Universal Robots PolyScope program: Programa_PickPlace.urp

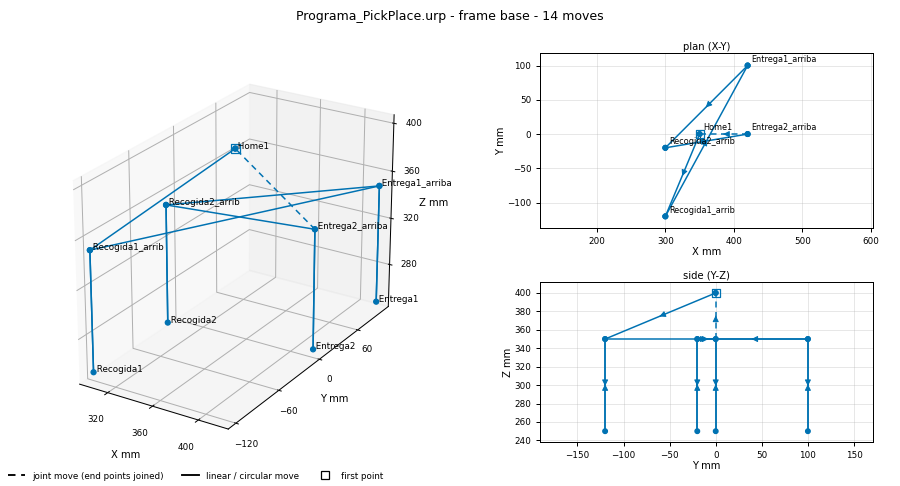
[picture p0: tool path of Programa_PickPlace.urp in frame base, 14 of 14 moves have a stored position in this frame; points joined in program order, loops and branches not executed]
Program Programa_PickPlace (installation=lab_manipulador directory=/ursim/programs createdIn=3.15.8.106339 lastSavedIn=3.15.8.106339 robotSerialNumber=2018359999)
Calibrated DH parameters: a=[0, -0.425, -0.39225, 0, 0, 0]; d=[0.089159, 0, 0, 0.10915, 0.09465, 0.0823]; alpha=[1.570796, 0, 0, 1.570796, -1.570796, 0]; deltaTheta=[0, 0, 0, 0, 0, 0]
Robot Program (runOnlyOnce=false)
  Set DigitalOutput (payload=0.5 tcpAsCog=true) pin=digital_out[0]; digitalValue=0
  MoveJ speed 60 deg/s, acceleration 80 deg/s^2 (useActiveTCP=true)
    Waypoint Home1: TCP in base x=350 y=0 z=400 mm, rx=0 ry=3.1412 rz=0 rad; joints [18.173, -68.7, -111.718, -89.559, 89.993, 108.173] deg
  MoveL speed 50 mm/s, acceleration 100 mm/s^2 (useActiveTCP=true) feature=Base
    Waypoint Recogida1_arrib: TCP in base x=300 y=-120 z=350 mm, rx=0 ry=-3.1412 rz=0 rad; joints [-2.058, -64.862, -121.221, -83.94, 89.999, 87.942] deg
    Waypoint Recogida1: TCP in base x=300 y=-120 z=250 mm, rx=0 ry=-3.1412 rz=0 rad; joints [-2.058, -69.151, -133.964, -66.908, 89.999, 87.942] deg
  Set DigitalOutput (payload=0.7 tcpAsCog=true) pin=digital_out[0]; digitalValue=1
  Wait Sleep waitTime=0.5
  MoveL speed 50 mm/s, acceleration 100 mm/s^2 (useActiveTCP=true) feature=Base
    Waypoint Recogida1_arrib: TCP in base x=300 y=-120 z=350 mm, rx=0 ry=-3.1412 rz=0 rad; joints [-2.058, -64.862, -121.221, -83.94, 89.999, 87.942] deg
    Waypoint Entrega1_arriba: TCP in base x=420 y=100 z=350 mm, rx=0 ry=-3.1412 rz=0 rad; joints [28.034, -81.687, -109.687, -78.646, 90.011, 118.034] deg
    Waypoint Entrega1: TCP in base x=420 y=100 z=250 mm, rx=0 ry=-3.1412 rz=0 rad; joints [28.034, -86.649, -120.847, -62.524, 90.011, 118.034] deg
  Set DigitalOutput (payload=0.5 tcpAsCog=true) pin=digital_out[0]; digitalValue=0
  Wait Sleep waitTime=0.5
  MoveL speed 50 mm/s, acceleration 100 mm/s^2 (useActiveTCP=true) feature=Base
    Waypoint Entrega1_arriba: TCP in base x=420 y=100 z=350 mm, rx=0 ry=-3.1412 rz=0 rad; joints [28.034, -81.687, -109.687, -78.646, 90.011, 118.034] deg
  MoveL speed 50 mm/s, acceleration 100 mm/s^2 (useActiveTCP=true) feature=Base
    Waypoint Recogida2_arrib: TCP in base x=300 y=-20 z=350 mm, rx=0 ry=-3.1412 rz=0 rad; joints [17.47, -61.06, -123.143, -85.819, 90.007, 107.47] deg
    Waypoint Recogida2: TCP in base x=300 y=-20 z=250 mm, rx=0 ry=-3.1412 rz=0 rad; joints [17.47, -64.911, -136.27, -68.842, 90.007, 107.47] deg
  Set DigitalOutput (payload=0.7 tcpAsCog=true) pin=digital_out[0]; digitalValue=1
  Wait Sleep waitTime=0.5
  MoveL speed 50 mm/s, acceleration 100 mm/s^2 (useActiveTCP=true) feature=Base
    Waypoint Recogida2_arrib: TCP in base x=300 y=-20 z=350 mm, rx=0 ry=-3.1412 rz=0 rad; joints [17.47, -61.06, -123.143, -85.819, 90.007, 107.47] deg
    Waypoint Entrega2_arriba: TCP in base x=420 y=0 z=350 mm, rx=0 ry=-3.1412 rz=0 rad; joints [15.062, -79.973, -111.099, -78.95, 90.006, 105.062] deg
    Waypoint Entrega2: TCP in base x=420 y=0 z=250 mm, rx=0 ry=-3.1412 rz=0 rad; joints [15.062, -84.942, -122.401, -62.679, 90.006, 105.062] deg
  Set DigitalOutput (payload=0.5 tcpAsCog=true) pin=digital_out[0]; digitalValue=0
  Wait Sleep waitTime=0.5
  MoveL speed 50 mm/s, acceleration 100 mm/s^2 (useActiveTCP=true) feature=Base
    Waypoint Entrega2_arriba: TCP in base x=420 y=0 z=350 mm, rx=0 ry=-3.1412 rz=0 rad; joints [15.062, -79.973, -111.099, -78.95, 90.006, 105.062] deg
  MoveJ speed 60 deg/s, acceleration 80 deg/s^2 (useActiveTCP=true)
    Waypoint Home1: TCP in base x=350 y=0 z=400 mm, rx=0 ry=3.1412 rz=0 rad; joints [18.173, -68.7, -111.718, -89.559, 89.993, 108.173] deg
  Wait DigitalInput pin=digital_in[0]; digitalValue=0
  Wait DigitalInput pin=digital_in[0]; digitalValue=1
